// TIA Portal V20 export
VAR_GLOBAL   // PLC tag table "ConvConstantA1"
END_VAR
VAR_GLOBAL CONSTANT   // user constants
   minA1 : Int := 1001;
   maxA1 : Int := 1002;
END_VAR
